INTERFACE I_Axis

PROPERTY Busy : BOOL
GET
END_GET
END_PROPERTY

PROPERTY Calibrated : BOOL
GET
END_GET
END_PROPERTY

PROPERTY Error : BOOL
GET
END_GET
END_PROPERTY

END_INTERFACE

(* stored: Version 1.1.0.1, ProductVersion 3.1.4026.11
   Itf I_Axis: Id {595a9217-864b-493b-b1f1-9dea5601aca8}
   Property Busy: Id {ba5504aa-3dda-42ca-bac2-51c45207c93a}
   Get Get: Id {b9cb56cd-c171-469f-b53d-6f00d1c9714f}
   Property Calibrated: Id {19e9d110-74bf-4045-a3bf-5f358d99765b}
   Get Get: Id {e5bd9191-9ec2-48a2-8d46-291347e47d6c}
   Property Error: Id {38bbb32e-3c0a-4087-ba48-cbebfbc23d31}
   Get Get: Id {fb98412b-4dc9-45ea-adcd-7d8dc14c2ef1} *)
